// TwinCAT 3 PLC project Main
// ProgramVersion: 3.1.4023.0
// libraries:
//   Tc2_Standard, * (Beckhoff Automation GmbH)
//   Tc2_System, * (Beckhoff Automation GmbH)
//   Tc3_Module, * (Beckhoff Automation GmbH)
//   VisuSymbols,3.5.10.0,System
// project tree:
//   / GlobalTextList.TcGTLO, PlcTask.TcTTO, 视图管理器.TcVMO (not stored)
//   GVLs/ GVL.TcGVL
//   POUs/ FB_StarDeltaStarter.TcPOU, MAIN.TcPOU
//   VISUs/ Visualization.TcVIS
// real-time tasks:
//   TASK PlcTask: cycle T#10ms, priority 20, ADS port 350

CONFIGURATION Main
    RESOURCE PLC ON TwinCAT3
        TASK PlcTask(INTERVAL := T#10ms, PRIORITY := 21);
        PROGRAM MAIN WITH PlcTask : MAIN;
    END_RESOURCE
END_CONFIGURATION

// ---- GVLs/GVL.TcGVL
{attribute 'qualified_only'}
VAR_GLOBAL
	iStartPB			: BOOL;
	iStopPB				: BOOL;
	iMainDelay			: TIME;
	iSwitchDelay		: TIME;
	
	oMainContactor		: BOOL;
	oStarContactor		: BOOL;
	oDeltaContactor		: BOOL;
	oState				: WSTRING;
END_VAR

// ---- POUs/MAIN.TcPOU
PROGRAM MAIN
VAR
	fbStarter		: FB_StarDeltaStarter;
END_VAR

fbStarter(
	bStart:= GVL.iStartPB, 
	bStop:= GVL.iStopPB, 
	tMainDelay:= T#1S, 
	tStarDeltaDelay:= T#5S, 
	bMainContactor=> GVL.oMainContactor, 
	bStarContactor=> GVL.oStarContactor, 
	bDeltaContactor=> GVL.oDeltaContactor,
	sStateDesciption => GVL.oState);

END_PROGRAM

// ---- POUs/FB_StarDeltaStarter.TcPOU
FUNCTION_BLOCK FB_StarDeltaStarter
VAR_INPUT
	bStart, bStop						: BOOL;
	tMainDelay							: TIME := T#1S;
	tStarDeltaDelay						: TIME := T#5S;
END_VAR
VAR_OUTPUT
	bMainContactor, bStarContactor, bDeltaContactor		: BOOL;
	sStateDesciption	: WSTRING;
	bActive				: BOOL;
	bBusy				: BOOL;
	bDone				: BOOL;
END_VAR
VAR
	_step				: INT := 0;
	_MainTimer			: TON;
	_StarDeltaTimer		: TON;
END_VAR

CASE _step OF
	0	:
		sStateDesciption := "Step 0 : init Finished!";
		bMainContactor := FALSE;
		bStarContactor := FALSE;
		bDeltaContactor := FALSE;
		_MainTimer(IN := FALSE);
		IF bStart THEN
			_step := 10;
		END_IF
	10	:
		IF bStop THEN
			_step := 0;
		END_IF
		sStateDesciption := "Step 10 : Main contactor ON then delay!";
		bMainContactor := TRUE;
		_MainTimer(IN := TRUE, PT := tMainDelay);
		IF _MainTimer.Q THEN
			_MainTimer(IN := FALSE);
			_step := 11;
		END_IF
	11	:
		sStateDesciption := "Step 11 : Main contactor ON, star contactor delay!";
		bStarContactor := TRUE;
		_StarDeltaTimer(IN := TRUE, PT := tStarDeltaDelay);
		IF _StarDeltaTimer.Q THEN
			_StarDeltaTimer(IN := FALSE);
			bStarContactor := FALSE;
			_step := 110;
		END_IF
		IF bStop THEN
			_StarDeltaTimer(IN := FALSE);
			bStarContactor := FALSE;
			_step := 13;
		END_IF
	110	:
		sStateDesciption := "Step 110 : Main contactor ON, switch delay!";
		_MainTimer(IN := TRUE, PT := T#1S);
		IF _MainTimer.Q THEN
			_MainTimer(IN := FALSE);
			_step := 12;
		END_IF
		IF bStop THEN
			_MainTimer(IN := FALSE);
			bStarContactor := FALSE;
			_step := 13;
		END_IF
	12	:
		sStateDesciption := "Step 12 : Main and delta contactor ON!";
		bDeltaContactor := TRUE;
		IF bStop THEN
			bDeltaContactor :=FALSE;
			_step := 13;
		END_IF
	13	:
		sStateDesciption := "Step 13 : Delta OFF, delay Main OFF!";
		_MainTimer(IN := TRUE, PT := tMainDelay);
		IF _MainTimer.Q THEN
			_MainTimer(IN := FALSE);
			_step := 0;
		END_IF
END_CASE


	bDone := _step = 12;
	bActive := NOT (_step = 0);
	bBusy := bActive;

END_FUNCTION_BLOCK

// ---- GlobalTextList.TcGTLO
TEXTLIST GlobalTextList
  715 = '%s'
  410 = 'GO'
  839 = 'Stop'
END_TEXTLIST

// ---- VISUs/Visualization.TcVIS
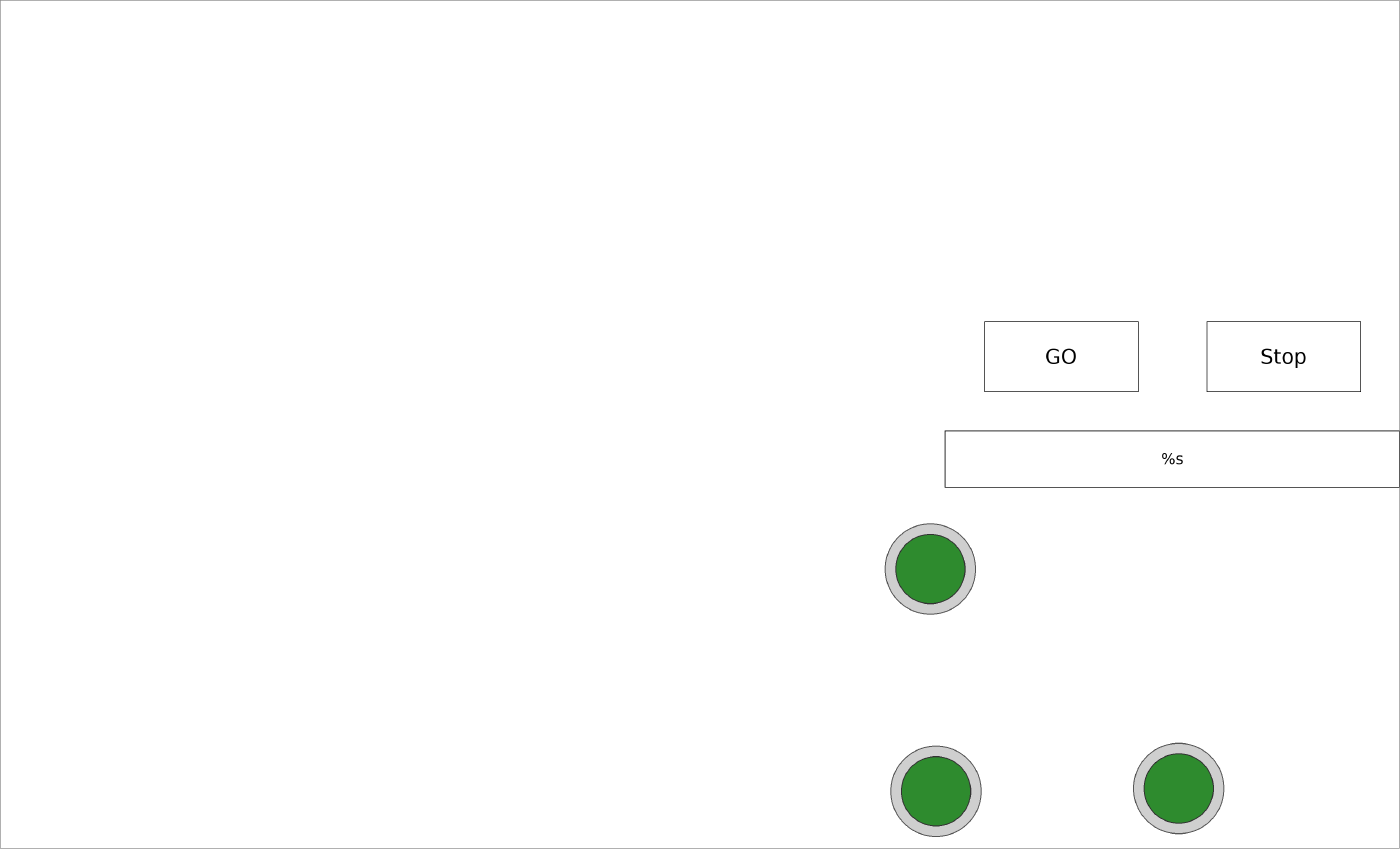
VISUALIZATION Visualization  // 1990x1207
    Lamp1 (1247,727 151x164), variable: GVL.oMainContactor, style: Lamp-Lamp1-Green
    Lamp1 (1600,1039 151x164), variable: GVL.oStarContactor, style: Lamp-Lamp1-Green
    Lamp1 (1255,1043 151x164), variable: GVL.oDeltaContactor, style: Lamp-Lamp1-Green
    Rectangle (1399,457 219x100), "GO"
        OnMouseDown: execute { GVL.iStartPB := true; }
        OnMouseUp: execute { GVL.iStartPB := false; }
    Rectangle (1715,457 219x100), "Stop"
        OnMouseDown: execute { GVL.iStopPB := true; }
        OnMouseUp: execute { GVL.iStopPB := false; }
    Rectangle (1343,612 647x81), "%s", text variable: GVL.oState
END_VISUALIZATION
